(* IEC 61131-3 sources: virtuepot/watertank/openplc, 1 file *)

(* ---- PLC1.st ---- *)
PROGRAM PLC1
  VAR
    level AT %IW0 : INT;
    Richiesta AT %QX0.2 : BOOL;
    request AT %IW1 : INT;
    pumps AT %QX0.0 : BOOL;
    valve AT %QX0.1 : BOOL;
    low AT %MX0.0 : BOOL;
    high AT %MX0.1 : BOOL;
    open_req AT %MX0.3 : BOOL;
    close_req AT %MX0.4 : BOOL;
    low_1 AT %MW0 : INT := 40;
    high_1 AT %MW1 : INT := 80;
  END_VAR
  VAR
    LE3_OUT : BOOL;
    GE7_OUT : BOOL;
  END_VAR

  LE3_OUT := LE(level, low_1);
  low := LE3_OUT;
  GE7_OUT := GE(level, high_1);
  high := GE7_OUT;
  open_req := Richiesta;
  close_req := NOT(Richiesta);
  pumps := NOT(high) AND (low OR pumps);
  valve := NOT(close_req) AND (open_req AND NOT(low) OR valve);
END_PROGRAM

CONFIGURATION Config0

  RESOURCE Res0 ON PLC
    TASK task0(INTERVAL := T#20ms,PRIORITY := 0);
    PROGRAM instance0 WITH task0 : PLC1;
  END_RESOURCE
END_CONFIGURATION
